// TIA Portal V18 export
TYPE "UDT_Marking CharToASCII"
// stored: IsFailsafeCompliant false
   STRUCT
      "Byte" : Array[0..127] of Byte;
   END_STRUCT;
END_TYPE
